# EPICS substitutions: current/app/Db/SystemAlarm.substitutions
file hpm900mbbiDirect.template {
  pattern {RECORD_NAME, OFFSET, FANOUT_RECORD}
  {SYSTEM_ALARM_RBV, 31, SYSTEM_ALARM_FANOUT}
}

file fanout15bit.template {
    pattern {RECORD_NAME,LINK0,LINK1,LINK2,LINK3,LINK4,LINK5,LINK6,LINK7,LINK8,LINK9,LINKA,LINKB,LINKC,LINKD,LINKE}
    {SYSTEM_ALARM_FANOUT,
     ALARM_RMT_SHUTDOWN_RBV,
     ALARM_EMO_BTN_PRESSED_RBV,
     ALARM_GAS_DET_WN_IN_RBV,
     ALARM_GAS_DET_ALM_IN_RBV,
     ALARM_FIRE_DET_IN_RBV,
     ALARM_COAX_IN_RBV,
     ALARM_EX_DP_SW_RBV,
     ALARM_N2_PRESS_SW_RBV,
     ALARM_Z_PURGE_PRESS_SW_RBV,
     ALARM_GAS_ON_IN_RBV,
     ALARM_DIG_IN_1_RBV,
     ALARM_DIG_IN_2_RBV,
     ALARM_DIG_IN_3_RBV,
     ALARM_DIG_IN_4_RBV,
     ALARM_SYST_STARTUP_RBV}
}

file hpm900bi.template {
    pattern {RECORD_NAME, DESC, BIT, INP}
    {ALARM_RMT_SHUTDOWN_RBV, "System Alarm, Remote Shutdown Triggered", 0, SYSTEM_ALARM_RBV}
    {ALARM_EMO_BTN_PRESSED_RBV, "System Alarm, EMO Button Pressed", 1, SYSTEM_ALARM_RBV}
    {ALARM_GAS_DET_WN_IN_RBV, "System Alarm, Gas Detector WN inp Trig", 2, SYSTEM_ALARM_RBV}
    {ALARM_GAS_DET_ALM_IN_RBV, "System Alarm, Gas Detector ALM inp Trig", 3, SYSTEM_ALARM_RBV}
    {ALARM_FIRE_DET_IN_RBV, "System Alarm, Fire Detector Input Trig", 4, SYSTEM_ALARM_RBV}
    {ALARM_COAX_IN_RBV, "System Alarm, COAX Input Triggered", 5, SYSTEM_ALARM_RBV}
    {ALARM_EX_DP_SW_RBV, "System Alarm, Exhaust DP Switch Trig", 6, SYSTEM_ALARM_RBV}
    {ALARM_N2_PRESS_SW_RBV, "System Alarm,N2 Pressure Switch Inp Trig", 7, SYSTEM_ALARM_RBV}
    {ALARM_Z_PURGE_PRESS_SW_RBV, "SysAlarm,Z Purge Pressure Switch InpTrig", 8, SYSTEM_ALARM_RBV}
    {ALARM_GAS_ON_IN_RBV, "System Alarm, Gas-On Input Triggered", 9, SYSTEM_ALARM_RBV}
    {ALARM_DIG_IN_1_RBV, "System Alarm, Digital Input 1 Triggered", A, SYSTEM_ALARM_RBV}
    {ALARM_DIG_IN_2_RBV, "System Alarm, Digital Input 2 Triggered", B, SYSTEM_ALARM_RBV}
    {ALARM_DIG_IN_3_RBV, "System Alarm, Digital Input 3 Triggered", C, SYSTEM_ALARM_RBV}
    {ALARM_DIG_IN_4_RBV, "System Alarm, Digital Input 4 Triggered", D, SYSTEM_ALARM_RBV}
    {ALARM_SYST_STARTUP_RBV, "System Alarm, System Start Up", E, SYSTEM_ALARM_RBV}

}
